FUNCTION "FBtest2" : Void
{ S7_Optimized_Access := 'TRUE' }
VERSION : 0.1
   VAR_INPUT
      bInput_mod : Bool;
   END_VAR


BEGIN
END_FUNCTION

